// SIMATIC STEP 7 (V5.x) project TEMA 8 EJERCICIO 5
// CPU: CPU313 C-2 DP(1)
// station: P_ADR_BUS
// station: Hardware
// station: Equipo SIMATIC 300
// program: Programa S7(1)

SYMBOL_TABLE
"FLANCOS"	DB 1	DB 1
"MANIOBRA"	DB 2	DB 2
"P PLANTA B"	I 0.0	BOOL
"P CABINA B"	I 0.1	BOOL
"P PLANTA 1"	I 0.2	BOOL
"P  CABINA 1"	I 0.3	BOOL
"FC PLANTA BAJA"	I 0.4	BOOL
"FC PLANTA 1"	I 0.5	BOOL
"Cycle Execution"	OB 1	OB 1
"S LENTA U1-V1-W1 RST"	Q 0.0	BOOL
"S RAPIDA U2-V2-W2 RST"	Q 0.1	BOOL
"CORTOCIRCUITADO SB"	Q 0.2	BOOL
"B LENTA U1-V1-W1 SRT"	Q 0.3	BOOL
"B RAPIDA U2-V2-W2 SRT"	Q 0.4	BOOL
"VAT_1"	VAT 1	
END_SYMBOL_TABLE

DATA_BLOCK "FLANCOS"	// DB 1
VERSION : 0.1
  STRUCT
   MARCA0 : BOOL ;
   MARCA1 : BOOL ;
   MARCA2 : BOOL ;
   MARCA3 : BOOL ;
   MARCA4 : BOOL ;
   MARCA5 : BOOL ;
   MARCA6 : BOOL ;
   MARCA7 : BOOL ;
   MARCA10 : BOOL ;
   MARCA11 : BOOL ;
   MARCA12 : BOOL ;
   MARCA13 : BOOL ;
   MARCA14 : BOOL ;
   MARCA15 : BOOL ;
   MARCA16 : BOOL ;
   MARCA17 : BOOL ;
  END_STRUCT ;	
BEGIN
END_DATA_BLOCK

DATA_BLOCK "MANIOBRA"	// DB 2
VERSION : 0.1
  STRUCT
   MARCA0 : BOOL ;
   MARCA1 : BOOL ;
   MARCA2 : BOOL ;
   MARCA3 : BOOL ;
   MARCA4 : BOOL ;
   MARCA5 : BOOL ;
   MARCA6 : BOOL ;
   MARCA7 : BOOL ;
  END_STRUCT ;	
BEGIN
END_DATA_BLOCK

ORGANIZATION_BLOCK "Cycle Execution"	// OB 1
TITLE = "Main Program Sweep (Cycle)"
//ACENSOR DE 2 PLANTAS CON MOTOR DHALANDER TEMPORIZADO EL CAMBIO DE VELOCIDAD
VERSION : 0.1
VAR_TEMP
  OB1_EV_CLASS : BYTE ;	//Bits 0-3 = 1 (Coming event), Bits 4-7 = 1 (Event class 1)
  OB1_SCAN_1 : BYTE ;	//1 (Cold restart scan 1 of OB 1), 3 (Scan 2-n of OB 1)
  OB1_PRIORITY : BYTE ;	//Priority of OB Execution
  OB1_OB_NUMBR : BYTE ;	//1 (Organization block 1, OB1)
  OB1_RESERVED_1 : BYTE ;	//Reserved for system
  OB1_RESERVED_2 : BYTE ;	//Reserved for system
  OB1_PREV_CYCLE : INT ;	//Cycle time of previous OB1 scan (milliseconds)
  OB1_MIN_CYCLE : INT ;	//Minimum cycle time of OB1 (milliseconds)
  OB1_MAX_CYCLE : INT ;	//Maximum cycle time of OB1 (milliseconds)
  OB1_DATE_TIME : DATE_AND_TIME ;	//Date and time OB1 started
END_VAR
BEGIN
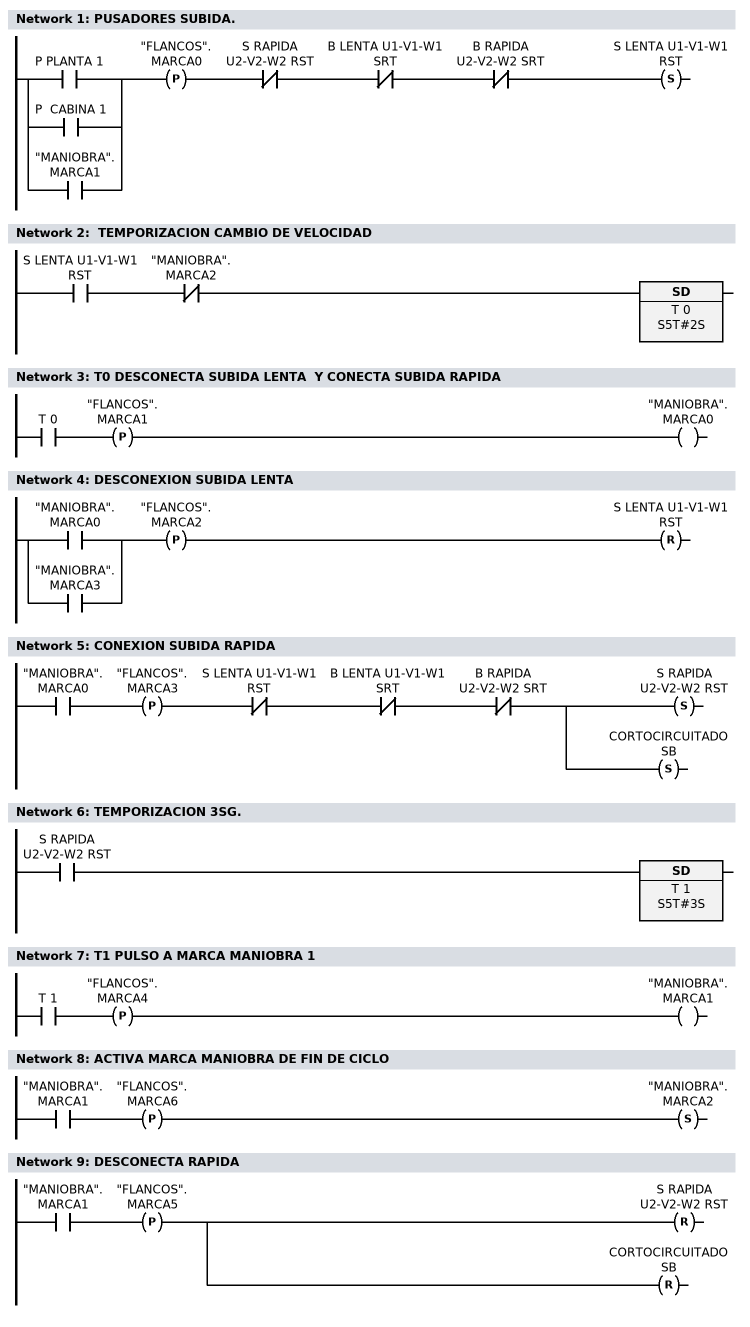
NETWORK
TITLE = PUSADORES SUBIDA. 
//LOS PULSADORES P. PLANTA 1 Y P CABINA 1 EJECUTARAN EL MISMO PROCESO YA QUE 
//EN LOS DOS CASOS EL ASCENSOR TIENE QUE SUBIR A LA PLANTA 1
//SUBIDA VELOCIDAD LENTA DURANTE 2 SEG.
      A(;
      O     "P PLANTA 1";
      O     "P  CABINA 1";
      O     "MANIOBRA".MARCA1;
      );
      FP    "FLANCOS".MARCA0;
      AN    "S RAPIDA U2-V2-W2 RST";
      AN    "B LENTA U1-V1-W1 SRT";
      AN    "B RAPIDA U2-V2-W2 SRT";
      S     "S LENTA U1-V1-W1 RST";
NETWORK
TITLE =  TEMPORIZACION CAMBIO DE VELOCIDAD
//ALIMENTACION TEMPORIZADOR SE 2SEG.
//
      A     "S LENTA U1-V1-W1 RST";
      AN    "MANIOBRA".MARCA2;
      L     S5T#2S;
      SD    T 0;
NETWORK
TITLE = T0 DESCONECTA SUBIDA LENTA  Y CONECTA SUBIDA RAPIDA
      A     T 0;
      FP    "FLANCOS".MARCA1;
      =     "MANIOBRA".MARCA0;
NETWORK
TITLE = DESCONEXION SUBIDA LENTA
      A(;
      O     "MANIOBRA".MARCA0;
      O     "MANIOBRA".MARCA3;
      );
      FP    "FLANCOS".MARCA2;
      R     "S LENTA U1-V1-W1 RST";
NETWORK
TITLE = CONEXION SUBIDA RAPIDA
      A     "MANIOBRA".MARCA0;
      FP    "FLANCOS".MARCA3;
      AN    "S LENTA U1-V1-W1 RST";
      AN    "B LENTA U1-V1-W1 SRT";
      AN    "B RAPIDA U2-V2-W2 SRT";
      S     "S RAPIDA U2-V2-W2 RST";
      S     "CORTOCIRCUITADO SB";
NETWORK
TITLE = TEMPORIZACION 3SG.
      A     "S RAPIDA U2-V2-W2 RST";
      L     S5T#3S;
      SD    T 1;
NETWORK
TITLE = T1 PULSO A MARCA MANIOBRA 1 
      A     T 1;
      FP    "FLANCOS".MARCA4;
      =     "MANIOBRA".MARCA1;
NETWORK
TITLE = ACTIVA MARCA MANIOBRA DE FIN DE CICLO
      A     "MANIOBRA".MARCA1;
      FP    "FLANCOS".MARCA6;
      S     "MANIOBRA".MARCA2;
NETWORK
TITLE = DESCONECTA RAPIDA 
      A     "MANIOBRA".MARCA1;
      FP    "FLANCOS".MARCA5;
      R     "S RAPIDA U2-V2-W2 RST";
      R     "CORTOCIRCUITADO SB";
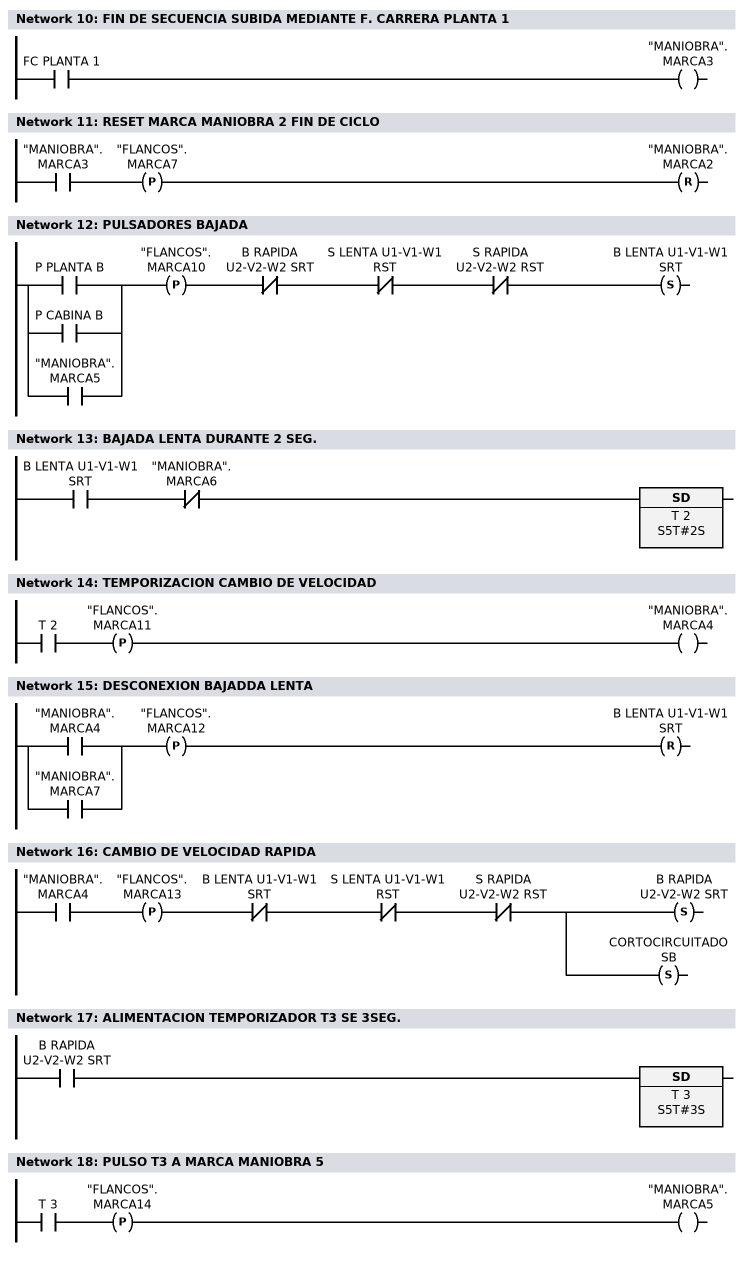
NETWORK
TITLE = FIN DE SECUENCIA SUBIDA MEDIANTE F. CARRERA PLANTA 1 
      A     "FC PLANTA 1";
      =     "MANIOBRA".MARCA3;
NETWORK
TITLE = RESET MARCA MANIOBRA 2 FIN DE CICLO
      A     "MANIOBRA".MARCA3;
      FP    "FLANCOS".MARCA7;
      R     "MANIOBRA".MARCA2;
NETWORK
TITLE = PULSADORES BAJADA
//LOS PULSADORES P PLANTA B Y P CABINA B EJECUTARAN EL MISMO PROCESO
//
      A(;
      O     "P PLANTA B";
      O     "P CABINA B";
      O     "MANIOBRA".MARCA5;
      );
      FP    "FLANCOS".MARCA10;
      AN    "B RAPIDA U2-V2-W2 SRT";
      AN    "S LENTA U1-V1-W1 RST";
      AN    "S RAPIDA U2-V2-W2 RST";
      S     "B LENTA U1-V1-W1 SRT";
NETWORK
TITLE = BAJADA LENTA DURANTE 2 SEG.
//ALIMENTACION TEMPORIZADOR T2 SE 2 SEG
      A     "B LENTA U1-V1-W1 SRT";
      AN    "MANIOBRA".MARCA6;
      L     S5T#2S;
      SD    T 2;
NETWORK
TITLE = TEMPORIZACION CAMBIO DE VELOCIDAD
//T2 DESCONECTA BAJADA LENTA Y CONECTA BAJADA RAPIDA
      A     T 2;
      FP    "FLANCOS".MARCA11;
      =     "MANIOBRA".MARCA4;
NETWORK
TITLE = DESCONEXION BAJADDA LENTA
      A(;
      O     "MANIOBRA".MARCA4;
      O     "MANIOBRA".MARCA7;
      );
      FP    "FLANCOS".MARCA12;
      R     "B LENTA U1-V1-W1 SRT";
NETWORK
TITLE = CAMBIO DE VELOCIDAD RAPIDA
      A     "MANIOBRA".MARCA4;
      FP    "FLANCOS".MARCA13;
      AN    "B LENTA U1-V1-W1 SRT";
      AN    "S LENTA U1-V1-W1 RST";
      AN    "S RAPIDA U2-V2-W2 RST";
      S     "B RAPIDA U2-V2-W2 SRT";
      S     "CORTOCIRCUITADO SB";
NETWORK
TITLE = ALIMENTACION TEMPORIZADOR T3 SE 3SEG.
      A     "B RAPIDA U2-V2-W2 SRT";
      L     S5T#3S;
      SD    T 3;
NETWORK
TITLE = PULSO T3 A MARCA MANIOBRA 5 
      A     T 3;
      FP    "FLANCOS".MARCA14;
      =     "MANIOBRA".MARCA5;
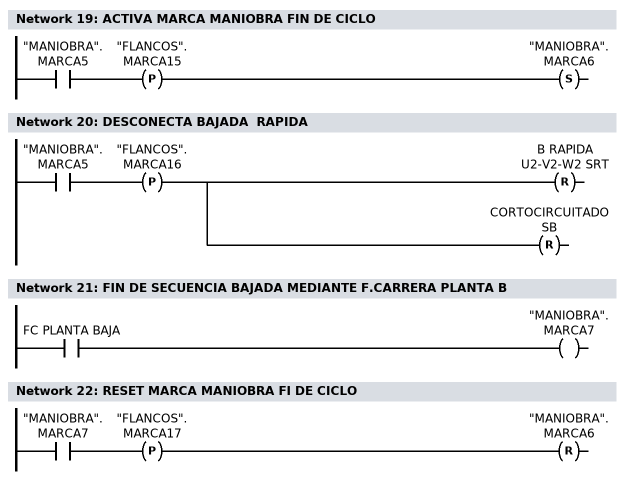
NETWORK
TITLE = ACTIVA MARCA MANIOBRA FIN DE CICLO
      A     "MANIOBRA".MARCA5;
      FP    "FLANCOS".MARCA15;
      S     "MANIOBRA".MARCA6;
NETWORK
TITLE = DESCONECTA BAJADA  RAPIDA
      A     "MANIOBRA".MARCA5;
      FP    "FLANCOS".MARCA16;
      R     "B RAPIDA U2-V2-W2 SRT";
      R     "CORTOCIRCUITADO SB";
NETWORK
TITLE = FIN DE SECUENCIA BAJADA MEDIANTE F.CARRERA PLANTA B
      A     "FC PLANTA BAJA";
      =     "MANIOBRA".MARCA7;
NETWORK
TITLE = RESET MARCA MANIOBRA FI DE CICLO
      A     "MANIOBRA".MARCA7;
      FP    "FLANCOS".MARCA17;
      R     "MANIOBRA".MARCA6;
END_ORGANIZATION_BLOCK
